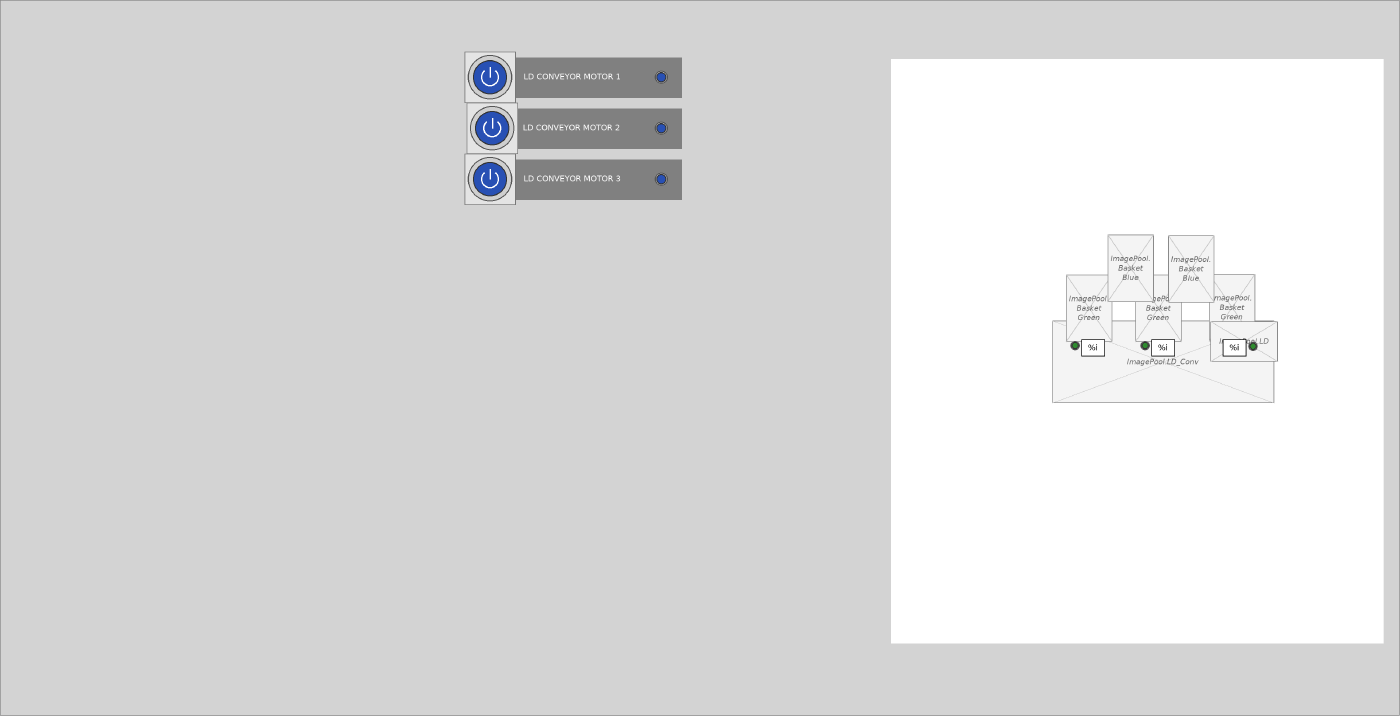
VISUALIZATION Manual_Loading  // 1920x983
    Rectangle (0,0 1920x983)
    Rectangle (1222,81 675x802)
    Image (1443,440 304x113), image: ImagePool.LD_Conv
    Image (1658,376 63x92), invisible if: NOT.ARbBasketGdFlag[1], image: ImagePool.Basket Green
        OnMouseDown: execute { AR2sDSCv_LdConfirmBasketInfo[1,3].iProductRecipeNo:=0; }
    Image (1462,377 63x92), invisible if: NOT AR2sDSCv_LdConfirmBasketInfo[1,1].bAvailibility, image: ImagePool.Basket Green
        OnMouseDown: execute { AR2sDSCv_LdConfirmBasketInfo[1,1].iProductRecipeNo:=0; }
    Image (1660,441 92x55), image: ImagePool.LD
    Image (1557,377 63x92), invisible if: NOT AR2sDSCv_LdConfirmBasketInfo[1,2].bAvailibility, image: ImagePool.Basket Green
        OnMouseDown: execute { AR2sDSCv_LdConfirmBasketInfo[1,2].iProductRecipeNo:=0; }
    Image (1519,322 63x92), invisible if: NOT AR2sDSCv_LdTransferBasketInfo[1,1].bAvailibility, image: ImagePool.Basket Blue
        OnMouseDown: execute { AR2sDSCv_LdTransferBasketInfo[1,1].iProductRecipeNo:=0; }
    Image (1602,323 63x92), invisible if: NOT AR2sDSCv_LdTransferBasketInfo[1,2].bAvailibility, image: ImagePool.Basket Blue
        OnMouseDown: execute { AR2sDSCv_LdTransferBasketInfo[1,2].iProductRecipeNo:=0;; }
    Lamp1 (1467,467 15x15), variable: ARdsMAP_HmiVariableGeneral.bLdFeedSensor_IND, style: Lamp-Lamp1-Green
    Lamp1 (1711,468 15x15), variable: ARdsMAP_HmiVariableGeneral.bLdPickSensor_IND, style: Lamp-Lamp1-Green
    RoundedRectangle (676,79 259x55)
    Label (715,91 176x29), "LD CONVEYOR MOTOR 1"
    Lamp1 (897,96 20x20), variable: ARdsMAP_HmiVariableGeneral.bLdConveyorMotor01_IND, style: Lamp-Lamp1-Blue
    PowerSwitch (637,71 70x70), variable: ARdsMAP_HmiVariableGeneral.bLdConveyorMotor01_PB, behaviour: TOGGLE, style: Switch-PowerSwitch-Blue
    RoundedRectangle (676,149 259x55)
    Label (714,161 178x29), "LD CONVEYOR MOTOR 2"
    Lamp1 (897,166 20x20), variable: ARdsMAP_HmiVariableGeneral.bLdConveyorMotor02_IND, style: Lamp-Lamp1-Blue
    PowerSwitch (640,141 70x70), variable: ARdsMAP_HmiVariableGeneral.bLdConveyorMotor02_PB, behaviour: TOGGLE, style: Switch-PowerSwitch-Blue
    RoundedRectangle (676,219 259x55)
    Label (715,231 176x29), "LD CONVEYOR MOTOR 3"
    Lamp1 (897,236 20x20), variable: ARdsMAP_HmiVariableGeneral.bLdConveyorMotor03_IND, style: Lamp-Lamp1-Blue
    PowerSwitch (637,211 70x70), variable: ARdsMAP_HmiVariableGeneral.bLdConveyorMotor03_PB, behaviour: TOGGLE, style: Switch-PowerSwitch-Blue
    Rectangle (1677,466 32x23), "%i", text variable: AR2sDSCv_LdConfirmBasketInfo[1,3].iProductRecipeNo
        OnMouseDown: write the text variable via VisuDialogs.Numpad
    Rectangle (1579,466 32x23), "%i", text variable: AR2sDSCv_LdConfirmBasketInfo[1,2].iProductRecipeNo
        OnMouseDown: write the text variable via VisuDialogs.Numpad
    Rectangle (1483,466 32x23), "%i", text variable: AR2sDSCv_LdConfirmBasketInfo[1,1].iProductRecipeNo
        OnMouseDown: write the text variable via VisuDialogs.Numpad
    Lamp1 (1563,467 15x15), variable: ARdsMAP_HmiVariableGeneral.bLdIndex1Sensor_IND, style: Lamp-Lamp1-Green
END_VISUALIZATION

(* stored: Version 1.1.0.1, ProductVersion 3.1.4024.12
   Visu Manual_Loading: Id {143bfa08-d81f-40f1-9d6f-90faca07e6fa} *)
